{attribute 'qualified_only'}
{attribute 'strict'}
{attribute 'to_string'}
TYPE E_Mode :
(
 	Idle := 0,
 	Homing,
 	Service,
 	Auto,
 	Error
)UINT;
END_TYPE

(* stored: Version 1.1.0.1, ProductVersion 3.1.4026.18
   DUT E_Mode: Id {538a5602-69d8-4e48-9192-e0c848920a4d} *)
